// TIA Portal V20 export
VAR_GLOBAL   // PLC tag table "Digital_Outputs"
   DQ_FreeQ0_0 AT %Q0.0 : Bool;
   DQ_OperatingCounter AT %Q0.1 : Bool;
   DQ_GeneralAirValve AT %Q0.2 : Bool;
   DQ_SmartLineDisable AT %Q0.3 : Bool;
   DQ_MachineLight AT %Q0.4 : Bool;
   DQ_MachineLightBack AT %Q0.5 : Bool;
   DQ_LightTowerOrange AT %Q0.6 : Bool;
   DQ_LightTowerRed AT %Q0.7 : Bool;
   DQ_LightTowerBlue AT %Q1.0 : Bool;
   DQ_Light_owerGreen AT %Q1.1 : Bool;
   DQ_LightTowerWhite AT %Q1.2 : Bool;
   DQ_Backlight AT %Q1.3 : Bool;
   DQ_FreeQ1_4 AT %Q1.4 : Bool;
   DQ_InfeedON AT %Q1.5 : Bool;
   DQ_AxisActivation AT %Q1.6 : Bool;
   DQ_BuzzerActivation AT %Q1.7 : Bool;
   DQ_ElbaronPowerON AT %Q2.0 : Bool;
   DQ_ObservationCameraLight AT %Q2.1 : Bool;
   DQ_LaserExternalDoorOpening AT %Q2.2 : Bool;
   DQ_CoolingStart AT %Q2.3 : Bool;
   DQ_X_AxisBrakeActivation AT %Q2.4 : Bool;
   DQ_Y_AxisBrakeActivation AT %Q2.5 : Bool;
   DQ_AxisB_TeachInClampingPart AT %Q2.6 : Bool;
   DQ_EPO_UPS AT %Q2.7 : Bool;
   DQ_HeadLaserStart AT %Q3.0 : Bool;
   DQ_HeadLaserStop AT %Q3.1 : Bool;
   DQ_Axis2_PowerContactor AT %Q3.2 : Bool;
   DQ_GasAssistOn AT %Q3.3 : Bool;
   DQ_SmartLineReset AT %Q3.4 : Bool;
   DQ_XY_AxisPowerContactor AT %Q3.5 : Bool;
   DQ_LaserAirPressureProcess AT %Q3.6 : Bool;
   DQ_Bus60V_PowerContactor AT %Q3.7 : Bool;
   DQ_FreeQ4_0 AT %Q4.0 : Bool;
   DQ_FreeQ4_1 AT %Q4.1 : Bool;
   DQ_FreeQ4_2 AT %Q4.2 : Bool;
   DQ_FreeQ4_3 AT %Q4.3 : Bool;
   DQ_LoadClampClosing AT %Q4.4 : Bool;
   DQ_LoadClampOpening AT %Q4.5 : Bool;
   DQ_UnloadClampClosing AT %Q4.6 : Bool;
   DQ_UnloadClampOpening AT %Q4.7 : Bool;
   DQ_ClampingOpening AT %Q5.0 : Bool;
   DQ_ClampingClosing AT %Q5.1 : Bool;
   DQ_B_AxisBrakeRelease AT %Q5.2 : Bool;
   DQ_Suction AT %Q5.3 : Bool;
   DQ_FreeQ5_4 AT %Q5.4 : Bool;
   DQ_FreeQ5_5 AT %Q5.5 : Bool;
   DQ_FreeQ5_6 AT %Q5.6 : Bool;
   DQ_FreeQ5_7 AT %Q5.7 : Bool;
   DQ_ExternalGateClosing AT %Q8.0 : Bool;
   DQ_ExternalGateOpening AT %Q8.1 : Bool;
   DQ_InternalGateClosing AT %Q8.2 : Bool;
   DQ_InternalGateOpening AT %Q8.3 : Bool;
   DQ_PowerMeterRetract AT %Q8.4 : Bool;
   DQ_PowerMeterAdvance AT %Q8.5 : Bool;
   DQ_Blowing AT %Q8.6 : Bool;   //    {ExternalWritable false}
   DQ_FreeQ8_7 AT %Q8.7 : Bool;
   DQ_FreeQ9_0 AT %Q9.0 : Bool;
   DQ_FreeQ9_1 AT %Q9.1 : Bool;
   DQ_FreeQ9_2 AT %Q9.2 : Bool;
   DQ_FreeQ9_3 AT %Q9.3 : Bool;
   DQ_FreeQ9_4 AT %Q9.4 : Bool;
   DQ_FreeQ9_5 AT %Q9.5 : Bool;
   DQ_FreeQ9_6 AT %Q9.6 : Bool;
   DQ_FreeQ9_7 AT %Q9.7 : Bool;
END_VAR
